{attribute 'linkalways'}
{attribute 'hide_all_locals'}
FUNCTION_BLOCK ValueDint EXTENDS ValueDintRead IMPLEMENTS Value
VAR
END_VAR

METHOD SetFromType : BOOL
VAR_INPUT
	source : __SYSTEM.AnyType;
END_VAR
SetFromType := ConvertAnyType(source, thisAnyType);
END_METHOD

METHOD SetFromString : BOOL
VAR_INPUT
	value : T_MaxString;
END_VAR
thisValue := STRING_TO_DINT(value);

SetFromString := TRUE;
END_METHOD

METHOD Set : BOOL
VAR_INPUT
	source : ANY;
END_VAR
Set := ConvertAnyType(source, thisAnyType);
END_METHOD

END_FUNCTION_BLOCK

(* stored: Version 1.1.0.1
   POU ValueDint: Id {6b5cc77d-0651-4d98-b1db-2c6fe535e4f0}, SpecialFunc None
   Method SetFromType: Id {f42f4189-5f01-413a-ab86-2686cf6e7d26}
   Method SetFromString: Id {c99ac060-1aa6-4527-aeaa-f5009ecc7633}
   Method Set: Id {cb0b1480-cfc4-4211-8b1a-8806afebd906} *)
